INTERFACE I_MessageData

PROPERTY DirRoot : POINTER to string(255)
SET
END_SET
END_PROPERTY

PROPERTY ErrorIndex : reference to uint
SET
END_SET
END_PROPERTY

PROPERTY FileRoot : pointer to string(255)
SET
END_SET
END_PROPERTY

PROPERTY LocalTime : pointer to DT
SET
END_SET
END_PROPERTY

PROPERTY MessageIndex : reference to uint
SET
END_SET
END_PROPERTY

PROPERTY MsgList : pointer to ARRAY[1..GVL_MSG_XTS.MAX_MESSAGE] OF st_message
SET
END_SET
END_PROPERTY

END_INTERFACE

(* stored: Version 1.1.0.1
   Itf I_MessageData: Id {6fee3d7d-7f98-4273-81c5-b0a80f56d680}
   Property DirRoot: Id {f8770dcc-e129-463e-a836-b4416642494d}
   Set Set: Id {9daafc0f-9e21-4d8e-96e9-abfa5e636c9d}
   Property ErrorIndex: Id {8b3d70fe-68c2-4483-8209-5ceb6a85bb6e}
   Set Set: Id {f149f307-053c-4723-b7de-2a6dac85b60e}
   Property FileRoot: Id {33a0e4aa-4b11-43a8-a509-795eab035a50}
   Set Set: Id {a5a75755-854f-4272-8bb6-bee5a6f894c6}
   Property LocalTime: Id {b2841289-08c3-475b-9d04-4f221d13138f}
   Set Set: Id {e88acbcc-949c-4bbb-94a8-9b82f5c836ce}
   Property MessageIndex: Id {cfc7cef0-1bab-4af2-a01f-8023b1fc13ab}
   Set Set: Id {0176821b-2abb-41d5-9ae4-6521b84223d9}
   Property MsgList: Id {ccd1ef7e-7618-45a0-9c85-867a3fd9fdc4}
   Set Set: Id {969a8b11-359f-47cb-8d5c-cc2d38816516} *)
